# EPICS substitutions: db/ecmcEL3164.substitutions
file ecmcEcSlave.template
{
    pattern {}
            {}
}

file ecmcEL3XXX-chX.template
{
	pattern {CH_ID, LINR,    ESLO,             EOFF,   EGU,        PREC, LOW, LOLO, HIGH, HIHI, HYST, LLSV,       LSV,        HSV,        HHSV      }
    		{1,     "SLOPE", 3.0518509476E-4,  0,      "V",        0,    0,   0,    0,    0,    0,    "NO_ALARM", "NO_ALARM", "NO_ALARM", "NO_ALARM"}
	    	{2,     "SLOPE", 3.0518509476E-4,  0,      "V",        0,    0,   0,    0,    0,    0,    "NO_ALARM", "NO_ALARM", "NO_ALARM", "NO_ALARM"}
		    {3,     "SLOPE", 3.0518509476E-4,  0,      "V",        0,    0,   0,    0,    0,    0,    "NO_ALARM", "NO_ALARM", "NO_ALARM", "NO_ALARM"}
		    {4,     "SLOPE", 3.0518509476E-4,  0,      "V",        0,    0,   0,    0,    0,    0,    "NO_ALARM", "NO_ALARM", "NO_ALARM", "NO_ALARM"}

}
